// Optional. Implement when a test needs preparation that may span scans and is

// worth separating from the body.

//

// The suite calls Setup to completion before the first call to Run. A failure or

// error recorded during setup ends the test without running the body - which is

// the point: a test whose fixture never came up has not been exercised, and

// reporting it as a failed check would be a lie.

//

// I_TestTiming.IsFirstCycle covers anything simpler than this.
INTERFACE I_TestSetup EXTENDS __SYSTEM.IQueryInterface

// Return TRUE when setup is complete. Enable behaves as in I_Test.Run.

//

// Bounded by its own deadline, separate from the test's.
METHOD Setup : BOOL
VAR_INPUT
	Enable : BOOL;
	Test   : I_TestAssertions;
END_VAR
END_METHOD

END_INTERFACE

(* stored: Version 1.1.0.1, ProductVersion 3.1.4026.18
   Itf I_TestSetup: Id {801db1ee-d024-43f8-a3f5-17427c23c39b}
   Method Setup: Id {83cf441f-77e4-427d-8089-ea8e8c02afed} *)
